(* Logix 5000 project; controller BreakGroup_US vendor 1 type 14 code 211 rev 32.16; software revision 32.05; part 8 of 8 *)
(* tags used below, declared in another part *)
   Emg_Stop : BOOL;
   HMI_MAN_STN_80_STOP : BOOL;
   HMI_MAN_STN_90_STOP : BOOL;
   MAN_STN_80_HOME : TIMER;
   MAN_STN_90_HOME : TIMER;
   MCP_ST_80_Turntable_Motor : MCP_Servo_02;
   RCP_ST_90_Turntable_Motor : RCP_Servo_02;
   ST10_Trolley1Lock_Cyl_01_Extended : ALIAS FOR MCP_PT01:1:I.0;
   ST_80_Start : BOOL;
   ST_90_Start : BOOL;
   STN_80_HMI_PB : SINT[2];
   STN_90_HMI_PB : SINT[2];

PROGRAM Station_80   (* main routine Main *)

ROUTINE Main   (* ladder *)
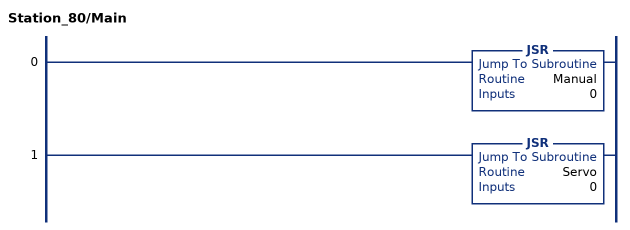
   0: JSR(Manual,0);
   1: JSR(Servo,0);
END_ROUTINE

ROUTINE Manual   (* ladder *)
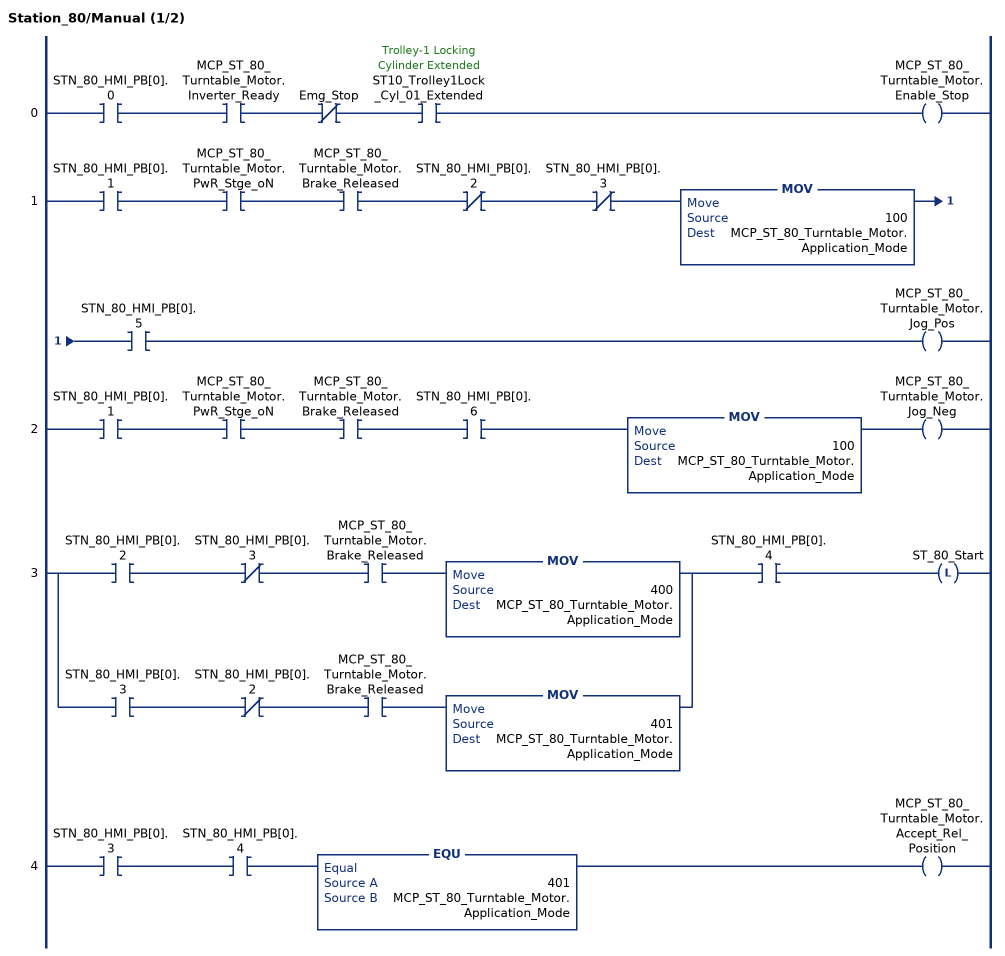
   0: XIC(STN_80_HMI_PB[0].0)XIC(MCP_ST_80_Turntable_Motor.Inverter_Ready)XIO(Emg_Stop)XIC(ST10_Trolley1Lock_Cyl_01_Extended)OTE(MCP_ST_80_Turntable_Motor.Enable_Stop);
   1: XIC(STN_80_HMI_PB[0].1)XIC(MCP_ST_80_Turntable_Motor.PwR_Stge_oN)XIC(MCP_ST_80_Turntable_Motor.Brake_Released)XIO(STN_80_HMI_PB[0].2)XIO(STN_80_HMI_PB[0].3)MOV(100,MCP_ST_80_Turntable_Motor.Application_Mode)XIC(STN_80_HMI_PB[0].5)OTE(MCP_ST_80_Turntable_Motor.Jog_Pos);
   2: XIC(STN_80_HMI_PB[0].1)XIC(MCP_ST_80_Turntable_Motor.PwR_Stge_oN)XIC(MCP_ST_80_Turntable_Motor.Brake_Released)XIC(STN_80_HMI_PB[0].6)MOV(100,MCP_ST_80_Turntable_Motor.Application_Mode)OTE(MCP_ST_80_Turntable_Motor.Jog_Neg);
   3: [XIC(STN_80_HMI_PB[0].2) XIO(STN_80_HMI_PB[0].3) XIC(MCP_ST_80_Turntable_Motor.Brake_Released) MOV(400,MCP_ST_80_Turntable_Motor.Application_Mode) ,XIC(STN_80_HMI_PB[0].3) XIO(STN_80_HMI_PB[0].2) XIC(MCP_ST_80_Turntable_Motor.Brake_Released) MOV(401,MCP_ST_80_Turntable_Motor.Application_Mode) ]XIC(STN_80_HMI_PB[0].4)OTL(ST_80_Start);
   4: XIC(STN_80_HMI_PB[0].3)XIC(STN_80_HMI_PB[0].4)EQU(401,MCP_ST_80_Turntable_Motor.Application_Mode)OTE(MCP_ST_80_Turntable_Motor.Accept_Rel_Position);
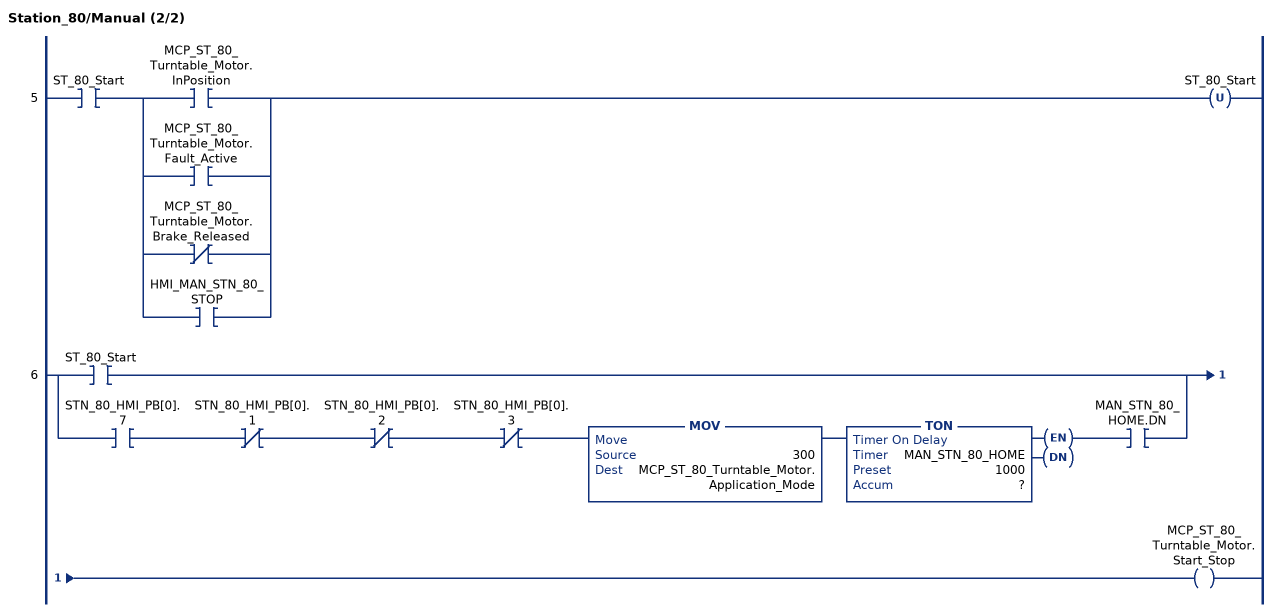
   5: XIC(ST_80_Start)[XIC(MCP_ST_80_Turntable_Motor.InPosition) ,[XIC(MCP_ST_80_Turntable_Motor.Fault_Active) ,[XIO(MCP_ST_80_Turntable_Motor.Brake_Released) ,XIC(HMI_MAN_STN_80_STOP) ] ] ]OTU(ST_80_Start);
   6: [XIC(ST_80_Start) ,XIC(STN_80_HMI_PB[0].7) XIO(STN_80_HMI_PB[0].1) XIO(STN_80_HMI_PB[0].2) XIO(STN_80_HMI_PB[0].3) MOV(300,MCP_ST_80_Turntable_Motor.Application_Mode) TON(MAN_STN_80_HOME,?,?) XIC(MAN_STN_80_HOME.DN) ]OTE(MCP_ST_80_Turntable_Motor.Start_Stop);
END_ROUTINE

ROUTINE Servo   (* ladder *)
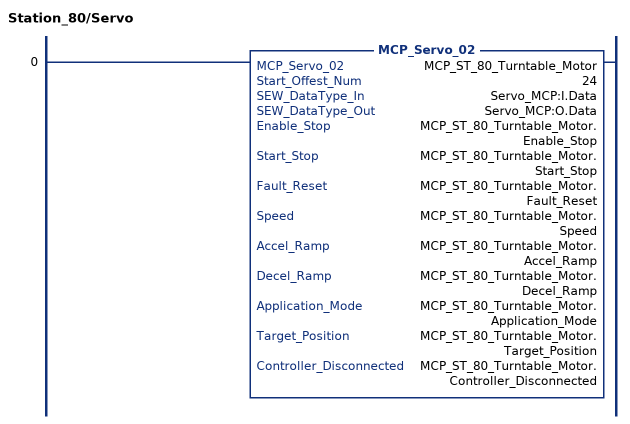
   0: MCP_Servo_02(MCP_ST_80_Turntable_Motor,24,Servo_MCP:I.Data,Servo_MCP:O.Data,MCP_ST_80_Turntable_Motor.Enable_Stop,MCP_ST_80_Turntable_Motor.Start_Stop,MCP_ST_80_Turntable_Motor.Fault_Reset,MCP_ST_80_Turntable_Motor.Speed,MCP_ST_80_Turntable_Motor.Accel_Ramp,MCP_ST_80_Turntable_Motor.Decel_Ramp,MCP_ST_80_Turntable_Motor.Application_Mode,MCP_ST_80_Turntable_Motor.Target_Position,MCP_ST_80_Turntable_Motor.Controller_Disconnected);
END_ROUTINE
END_PROGRAM

PROGRAM Station_90   (* main routine Main *)

ROUTINE Main   (* ladder *)
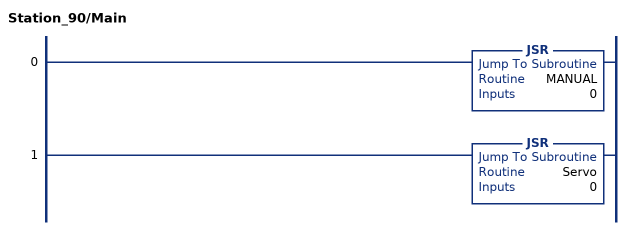
   0: JSR(MANUAL,0);
   1: JSR(Servo,0);
END_ROUTINE

ROUTINE MANUAL   (* ladder *)
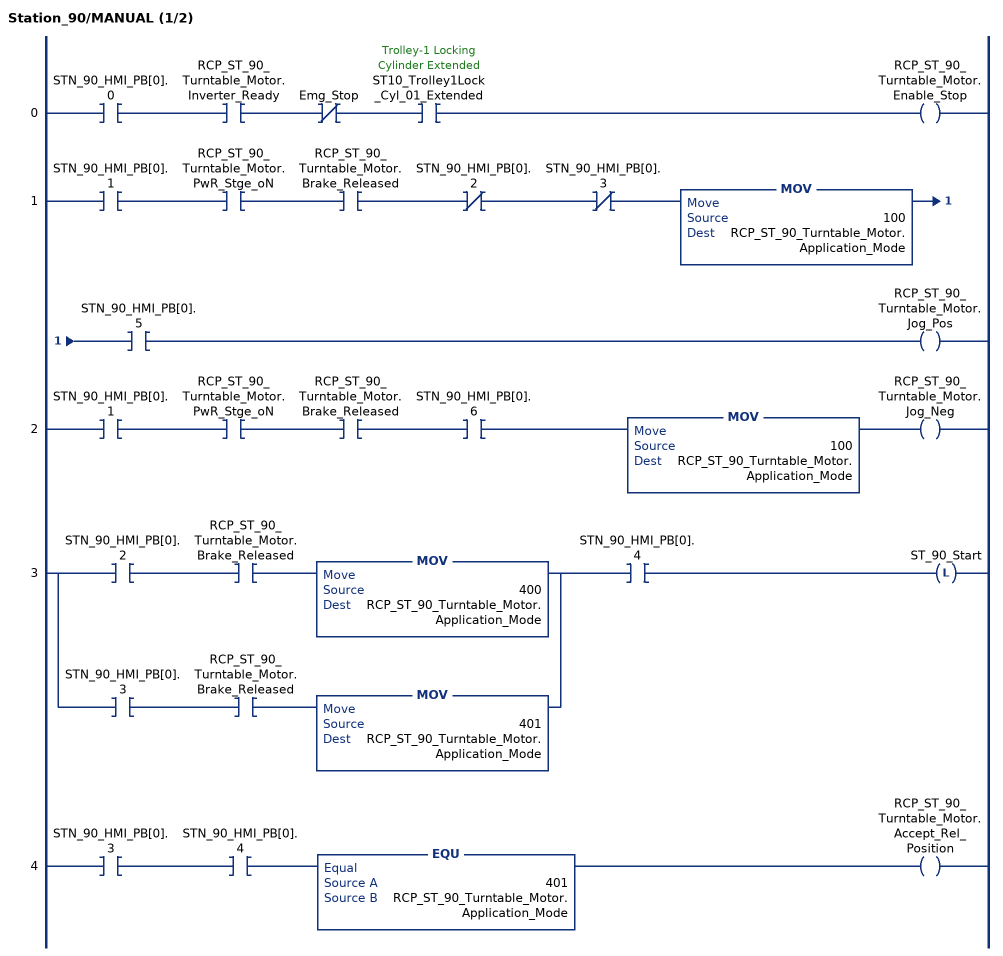
   0: XIC(STN_90_HMI_PB[0].0)XIC(RCP_ST_90_Turntable_Motor.Inverter_Ready)XIO(Emg_Stop)XIC(ST10_Trolley1Lock_Cyl_01_Extended)OTE(RCP_ST_90_Turntable_Motor.Enable_Stop);
   1: XIC(STN_90_HMI_PB[0].1)XIC(RCP_ST_90_Turntable_Motor.PwR_Stge_oN)XIC(RCP_ST_90_Turntable_Motor.Brake_Released)XIO(STN_90_HMI_PB[0].2)XIO(STN_90_HMI_PB[0].3)MOV(100,RCP_ST_90_Turntable_Motor.Application_Mode)XIC(STN_90_HMI_PB[0].5)OTE(RCP_ST_90_Turntable_Motor.Jog_Pos);
   2: XIC(STN_90_HMI_PB[0].1)XIC(RCP_ST_90_Turntable_Motor.PwR_Stge_oN)XIC(RCP_ST_90_Turntable_Motor.Brake_Released)XIC(STN_90_HMI_PB[0].6)MOV(100,RCP_ST_90_Turntable_Motor.Application_Mode)OTE(RCP_ST_90_Turntable_Motor.Jog_Neg);
   3: [XIC(STN_90_HMI_PB[0].2) XIC(RCP_ST_90_Turntable_Motor.Brake_Released) MOV(400,RCP_ST_90_Turntable_Motor.Application_Mode) ,XIC(STN_90_HMI_PB[0].3) XIC(RCP_ST_90_Turntable_Motor.Brake_Released) MOV(401,RCP_ST_90_Turntable_Motor.Application_Mode) ]XIC(STN_90_HMI_PB[0].4)OTL(ST_90_Start);
   4: XIC(STN_90_HMI_PB[0].3)XIC(STN_90_HMI_PB[0].4)EQU(401,RCP_ST_90_Turntable_Motor.Application_Mode)OTE(RCP_ST_90_Turntable_Motor.Accept_Rel_Position);
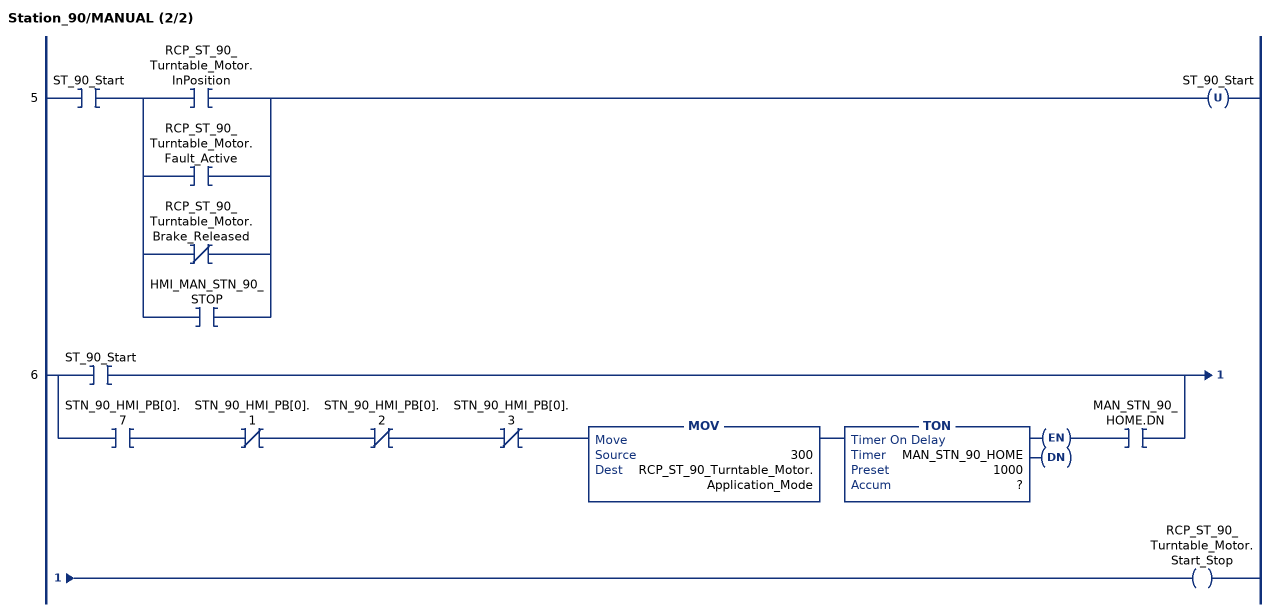
   5: XIC(ST_90_Start)[XIC(RCP_ST_90_Turntable_Motor.InPosition) ,[XIC(RCP_ST_90_Turntable_Motor.Fault_Active) ,[XIO(RCP_ST_90_Turntable_Motor.Brake_Released) ,XIC(HMI_MAN_STN_90_STOP) ] ] ]OTU(ST_90_Start);
   6: [XIC(ST_90_Start) ,XIC(STN_90_HMI_PB[0].7) XIO(STN_90_HMI_PB[0].1) XIO(STN_90_HMI_PB[0].2) XIO(STN_90_HMI_PB[0].3) MOV(300,RCP_ST_90_Turntable_Motor.Application_Mode) TON(MAN_STN_90_HOME,?,?) XIC(MAN_STN_90_HOME.DN) ]OTE(RCP_ST_90_Turntable_Motor.Start_Stop);
END_ROUTINE

ROUTINE Servo   (* ladder *)
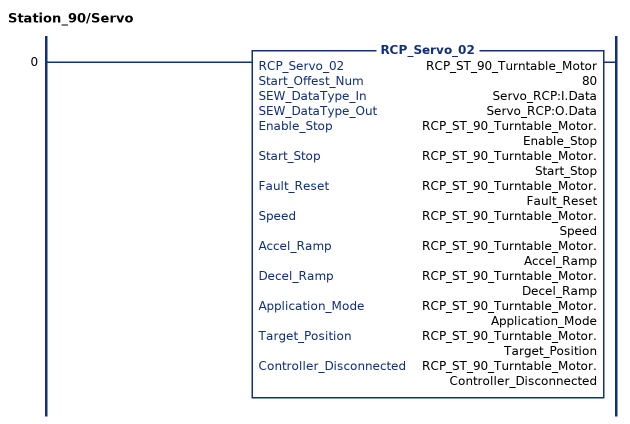
   0: RCP_Servo_02(RCP_ST_90_Turntable_Motor,80,Servo_RCP:I.Data,Servo_RCP:O.Data,RCP_ST_90_Turntable_Motor.Enable_Stop,RCP_ST_90_Turntable_Motor.Start_Stop,RCP_ST_90_Turntable_Motor.Fault_Reset,RCP_ST_90_Turntable_Motor.Speed,RCP_ST_90_Turntable_Motor.Accel_Ramp,RCP_ST_90_Turntable_Motor.Decel_Ramp,RCP_ST_90_Turntable_Motor.Application_Mode,RCP_ST_90_Turntable_Motor.Target_Position,RCP_ST_90_Turntable_Motor.Controller_Disconnected);
END_ROUTINE
END_PROGRAM
